{region '#Template'}
	{attribute 'Version' := '1.2.0.0'}
	{attribute 'Tags' := '"LCID": "1031", "Text": "General, Settings, Parameters, Basics"'}
	{attribute 'Tags' := '"LCID": "1033", "Text": "General, Settings, Parameters, Basics"'}
	{attribute 'Description' := '"LCID": "1031", "Text": "Basis Parameter für die Templates"'}
	{attribute 'Description' := '"LCID": "1033", "Text": "Basic parameters for the templates"'}
{endregion}
FUNCTION_BLOCK FB_BA_Settings EXTENDS FB_BA_View
VAR_INPUT
	fTWth					: REAL;	//	Weather temperature
END_VAR
VAR_INPUT CONSTANT
	WthParam			: FB_BA_WeatherParamter;
END_VAR
VAR

	GeneralSettings			: FB_BA_RawPublisher;									
	stSettings				: ST_BA_GeneralSettings;
END_VAR
VAR // added by the converter: edge detectors and wires of the graphical bodies
    _s1 : ST_BA_GeneralSettings;
END_VAR

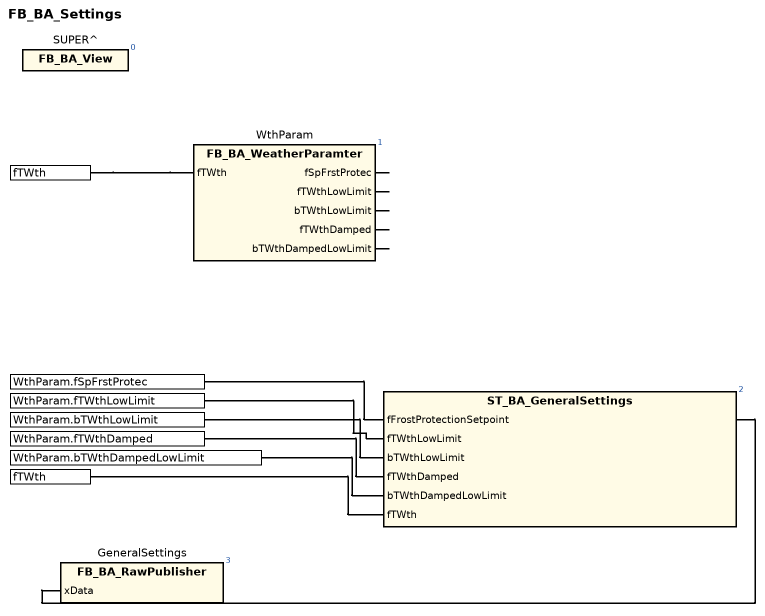
SUPER^(); // FB_BA_View
WthParam(fTWth := fTWth); // FB_BA_WeatherParamter
// compose _s1 : ST_BA_GeneralSettings
_s1.fFrostProtectionSetpoint := WthParam.fSpFrstProtec;
_s1.fTWthLowLimit := WthParam.fTWthLowLimit;
_s1.bTWthLowLimit := WthParam.bTWthLowLimit;
_s1.fTWthDamped := WthParam.fTWthDamped;
_s1.bTWthDampedLowLimit := WthParam.bTWthDampedLowLimit;
_s1.fTWth := fTWth;
GeneralSettings(xData := _s1); // FB_BA_RawPublisher

METHOD FB_init : BOOL
VAR_INPUT
	bInitRetains : BOOL; // if TRUE, the retain variables are initialized (warm start / cold start)
	bInCopyCode : BOOL;  // if TRUE, the instance afterwards gets moved into the copy code (online change)
END_VAR
WthParam.iParent				:= THIS^;
WthParam.iLabel					:= LblCmpGeneral.Settings_WthParam;
WthParam.sObjectName			:= '{Idx=01}';
WthParam.eDPADMode				:= E_BA_DPADMode.eInclude;
END_METHOD

END_FUNCTION_BLOCK

(* stored: Version 1.1.0.1, ProductVersion 3.1.4024.9
   POU FB_BA_Settings: Id {d7de45f0-e8dc-4b95-a8ac-ca86c9fe1868}, SpecialFunc None
   Method FB_init: Id {0b54a44c-2ead-49fe-9351-0a5dfac48d15} *)
